// TIA Portal project "PID_Tank_0" (V20)

(* hardware
DEVICE "S7-1500/ET200MP-Station_1"  S7-1500 station
   slot 0: "Profilschiene_0"  Rack  6ES7 590-1***0-0AA0
   slot 1: "PLC_1"  CPU 1515-2 PN  6ES7 515-2AM02-0AB0  V2.9
      slot 3: "CPU-Display_1"  6ES7591-1BA00-0AA0
      slot 32768: "PROFINET-Schnittstelle_1"  X1
         slot 32769: "Port_1"  X1 P1
         slot 32770: "Port_2"  X1 P2
      slot 33024: "PROFINET-Schnittstelle_2"  X2
         slot 33025: "Port_1"  X2 P1
      slot 34817: "Virtual CP interface port_1"  Virtual CP interface port  Virtual CP interface port
   slot 2: "DI 16x24VDC BA_1"  DI 16x24VDC BA  6ES7 521-1BH10-0AA0  V1.1
   slot 3: "DQ 16x24VDC/0.5A BA_1"  DQ 16x24VDC/0.5A BA  6ES7 522-1BH10-0AA0  V1.1
   slot 4: "AI 8xU/I/R/RTD BA_1"  AI 8xU/I/R/RTD BA  6ES7 531-7QF00-0AB0  V1.0
   slot 5: "AQ 8xU/I HS_1"  AQ 8xU/I HS  6ES7 532-5HF00-0AB0  V2.2
*)

// ===== PLC "PLC_1"  CPU 1515-2 PN =====

VAR_GLOBAL   // PLC tag table "Ausgaenge"
   "1M1" AT %QW30 : Int;   // Ventil Zufluss
   "2M1" AT %QW32 : Int;   // Ventil Abfluss
   "D1" AT %QW34 : Int;   // Anzeige Ist-Wert
   "D2" AT %AW36 : Int;   // Anzeige Soll-Wert
   "H1" AT %Q0.0 : Bool;   // Leuchte Füllen
   "H2" AT %Q0.1 : Bool;   // Leuchte Ablassen
END_VAR

VAR_GLOBAL   // PLC tag table "Eingaenge"
   "S1" AT %I0.0 : Bool;   // Füllen Taster
   "S2" AT %I0.1 : Bool;   // Ablassen Taster
   "FACTORY I/O (Running)" AT %I0.7 : Bool;
   "1B1" AT %IW30 : Int;   // Tank Füllhöhe
   "2B1" AT %EW32 : Int;   // Auslass Menge
   "1B2" AT %EW34 : Int;   // Tankeinstellung Soll-Wert
END_VAR

TYPE "typEingaenge"
   STRUCT
      S1 : Bool;   // Füllen Taster
      S2 : Bool;   // Ablassen Taster
      "1B1" : Int;   // Tank Füllhöhe
      "2B1" : Int;   // Auslass Menge
      "1B2" : Int;   // Tankeinstellung Soll-Wert
   END_STRUCT;
END_TYPE

TYPE "typAusgaenge"
   STRUCT
      H1 : Bool;   // Leuchte Füllen
      H2 : Bool;   // Leuchte Ablassen
      "1M1" : Int;   // Ventil Zufluss
      "2M1" : Int;   // Ventil Abfluss
      D1 : Int;   // Anzeige Ist-Wert
      D2 : Int;   // Anzeige Soll-Wert
   END_STRUCT;
END_TYPE

DATA_BLOCK "IDB_Anlage_ein"   // DB10
{ S7_Optimized_Access := 'TRUE' }
VERSION : 0.1
// stored: InstanceOfName Anlage_ein
"Anlage_ein"
BEGIN
END_DATA_BLOCK

DATA_BLOCK "HMI"   // DB100
{ S7_Optimized_Access := 'TRUE' }
VERSION : 0.1
   VAR
      Eingaenge : "typEingaenge";
      Ausgaenge : "typAusgaenge";
      Anlagedaten : Struct
         Sollmenge_cm : Real;
         Istmenge_cm : Real;
         Durchsatz_Abfluss_prozent : Real;
         Fuellstand_cm : Real;
         Tank_Volumen : Real;
         Stellwert_Ventil_fuellen : Real;
         Stellwert_Ventil_leeren : Real;
         Tank_leeren : Bool;
      END_STRUCT;
   END_VAR
BEGIN
END_DATA_BLOCK

FUNCTION_BLOCK "Anlage_ein"   // FB10, FBD
{ S7_Optimized_Access := 'TRUE' }
VERSION : 0.1
   VAR
      MI_FTRIG_S1 : F_TRIG;
      MI_FTRIG_S2 : F_TRIG;
   END_VAR
BEGIN

REGION Network 1 (SCL): Eingänge erfassen
   "HMI".Eingaenge."S1" := "S1";
   "HMI".Eingaenge."S2" := "S2";
   "HMI".Eingaenge."1B1" := "1B1";
   "HMI".Eingaenge."2B1" := "2B1";
   "HMI".Eingaenge."1B2" := "1B2";
END_REGION

REGION Network 2 (SCL): Flanken
   #MI_FTRIG_S1(CLK:="S1");
   #MI_FTRIG_S2(CLK:="S2");
END_REGION
END_FUNCTION_BLOCK

FUNCTION "Anlage_aus" : Void   // FC10, FBD
{ S7_Optimized_Access := 'TRUE' }
VERSION : 0.1
BEGIN

REGION Network 1 (SCL): Leuchte Füllen
   "H1" := "HMI".Ausgaenge.H1;
   "H2" := "HMI".Ausgaenge.H2;
   "1M1" := "HMI".Ausgaenge."1M1";
   "2M1" := "HMI".Ausgaenge."2M1";
   "D1" := "HMI".Ausgaenge.D1;
   "D2" := "HMI".Ausgaenge.D2;
END_REGION
END_FUNCTION

FUNCTION "FC_Tank" : Void   // FC20, FBD
{ S7_Optimized_Access := 'TRUE' }
VERSION : 0.1
   VAR_TEMP
      Hoehe_temp : Real;
      Durchlass_temp : Real;
      Poti_temp : Real;
   END_VAR
BEGIN

REGION Network 1 (SCL): Skalierung der Werte
   // Fuellhoehe (Ist-Wert)
   #Hoehe_temp := NORM_X(MIN := 0, VALUE := "HMI".Eingaenge."1B1", MAX := 27648);
   "HMI".Anlagedaten.Istmenge_cm := SCALE_X(MIN := 0.0, VALUE := #Hoehe_temp, MAX := 300.0);

   // Abfluss (Ventil-Durchlass-Menge)
   #Durchlass_temp := NORM_X(MIN := 0, VALUE := "HMI".Eingaenge."2B1", MAX := 27648);
   "HMI".Anlagedaten.Durchsatz_Abfluss_prozent := SCALE_X(MIN := 0.0, VALUE := #Durchlass_temp, MAX := 100.0);

   // Potentiometer (Soll-Wert)
   #Poti_temp := NORM_X(MIN := 0, VALUE := "HMI".Eingaenge."1B2", MAX := 27648);
   "HMI".Anlagedaten.Sollmenge_cm := SCALE_X(MIN := 0.0, VALUE := #Poti_temp, MAX := 300.0);
END_REGION

REGION Network 3 (SCL): Werte für Display
   // Display (Ist-Wert)
   "HMI".Ausgaenge.D1 := REAL_TO_INT("HMI".Anlagedaten.Istmenge_cm);
   // Display (Soll-Wert)
   "HMI".Ausgaenge.D2 := REAL_TO_INT("HMI".Anlagedaten.Sollmenge_cm);
END_REGION
END_FUNCTION

FUNCTION "FC_Tanksteuerung" : Void   // FC21, FBD
{ S7_Optimized_Access := 'TRUE' }
VERSION : 0.1
   VAR_INPUT
      RTRIG_fuellen : Bool;
      RTRIG_leeren : Bool;
   END_VAR
   VAR_IN_OUT
      Tank_leeren : Bool;
   END_VAR
BEGIN

REGION Network 1 (SCL)
   IF #RTRIG_fuellen THEN
       ;
   END_IF;
END_REGION

REGION Network 2 (SCL)
   IF #RTRIG_leeren THEN
       #Tank_leeren := TRUE;
   END_IF;

   IF #Tank_leeren THEN

       IF "HMI".Anlagedaten.Fuellstand_cm <= 0.5 THEN
           #Tank_leeren := FALSE;
       END_IF;
   END_IF;
END_REGION
END_FUNCTION

ORGANIZATION_BLOCK "Main"   // OB1, FBD, ProgramCycle
TITLE = "Main Program Sweep (Cycle)"
{ S7_Optimized_Access := 'TRUE' }
VERSION : 0.1
   VAR_INPUT
      Initial_Call : Bool;   // Initial call of this OB
      Remanence : Bool;   // =True, if remanent data are available
   END_VAR
BEGIN

REGION Network 1
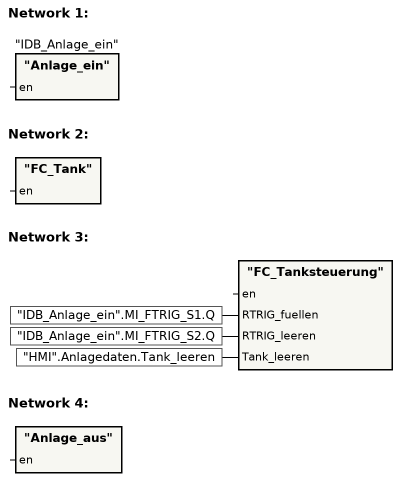
   "IDB_Anlage_ein"();   // "Anlage_ein"
END_REGION

REGION Network 2
   "FC_Tank"();
END_REGION

REGION Network 3
   "FC_Tanksteuerung"(RTRIG_fuellen := "IDB_Anlage_ein".MI_FTRIG_S1.Q,
                      RTRIG_leeren := "IDB_Anlage_ein".MI_FTRIG_S2.Q,
                      Tank_leeren := "HMI".Anlagedaten.Tank_leeren);
END_REGION

REGION Network 4
   "Anlage_aus"();
END_REGION
END_ORGANIZATION_BLOCK

ORGANIZATION_BLOCK "CyclicInterrupt"   // OB30, FBD, CyclicInterrupt
{ S7_Optimized_Access := 'TRUE' }
VERSION : 0.1
   VAR_INPUT
      Initial_Call : Bool;   // Initial call of this OB
      Event_Count : Int;   // Events discarded
   END_VAR
BEGIN

REGION Network 1
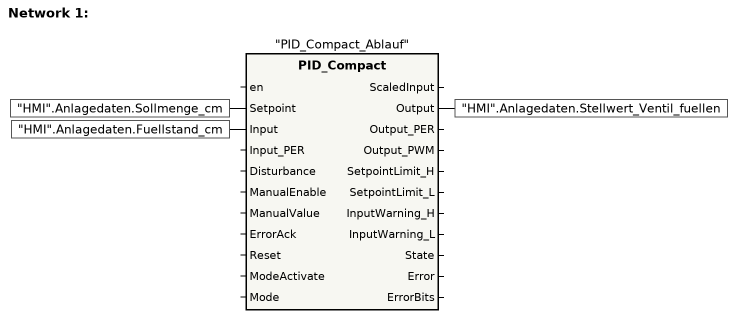
   "PID_Compact_Ablauf"(Setpoint := "HMI".Anlagedaten.Sollmenge_cm,   // PID_Compact
                        Input := "HMI".Anlagedaten.Fuellstand_cm,
                        Output => "HMI".Anlagedaten.Stellwert_Ventil_fuellen);
END_REGION
END_ORGANIZATION_BLOCK